Universal Robots PolyScope program: reciprocal_p3_3.urp

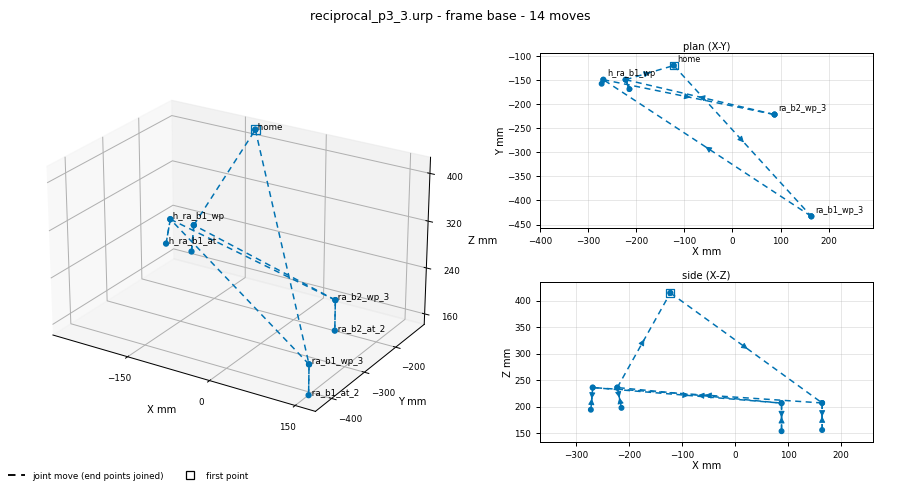
[picture p0: tool path of reciprocal_p3_3.urp in frame base, 14 of 14 moves have a stored position in this frame; points joined in program order, loops and branches not executed]
Program reciprocal_p3_3 (installation=default_1 directory=/programs/../media/urmountpoint_GSJLiG/ITER createdIn=5.3.1.64192 lastSavedIn=5.3.1.64192 robotSerialNumber=20195300365)
Calibrated DH parameters: a=[-0.000093, -0.190649, -0.212673, 0.000091, -0.000205, 0]; d=[0.151591, 44.061648, -42.488068, -1.442789, 0.085322, 0.091911]; alpha=[1.570082, -0.003447, 0.007513, 1.572293, -1.571904, 0]; deltaTheta=[0, -0.672656, 0.728185, -0.055522, 0.000005, 0]
Robot Program (runOnlyOnce=false)
  URCap Gripper Activate (Robotiq_Grippers, Robotiq Inc.) dataModel(ResetAndActivateKey=false)
  URCap Gripper (Robotiq_Grippers, Robotiq Inc.) dataModel(position=50.0, force=100.0, speed=100.0, positionInDouble=50.0, forceInDouble=100.0, speedInDouble=100.0, slaveIds=[9], blocking=true)
  MoveJ speed 60 deg/s, acceleration 80 deg/s^2 (useActiveTCP=true) feature=Base
    Waypoint home: TCP in base x=-122.15 y=-119.32 z=414.454 mm, rx=2.2563 ry=2.1459 rz=-0.0481 rad; joints [-85.681, -56.776, -79.802, -131.025, 89.944, -262.833] deg
  Folder Roof_A
    MoveJ speed 60 deg/s, acceleration 80 deg/s^2 (useActiveTCP=true) feature=Base
      Waypoint ra_b1_wp_3: TCP in base x=164.04 y=-432.993 z=207.005 mm, rx=2.2314 ry=2.1509 rz=0.0059 rad; joints [-53.036, -127.512, -66.191, -73.855, 90.777, -230.696] deg
      Waypoint ra_b1_at_2: TCP in base x=164.049 y=-432.987 z=156.003 mm, rx=2.2314 ry=2.151 rz=0.0059 rad; joints [-53.052, -131.715, -73.279, -62.563, 90.747, -230.647] deg
      URCap Gripper (Robotiq_Grippers, Robotiq Inc.) dataModel(position=100.0, force=100.0, speed=100.0, positionInDouble=100.0, forceInDouble=100.0, speedInDouble=100.0, slaveIds=[9], blocking=true)
      Waypoint ra_b1_wp_4: TCP in base x=164.04 y=-432.993 z=207.005 mm, rx=2.2314 ry=2.1509 rz=0.0059 rad; joints [-53.036, -127.512, -66.191, -73.855, 90.777, -230.696] deg
      Waypoint h_ra_b1_wp: TCP in base x=-268.55 y=-148.787 z=236.04 mm, rx=2.7608 ry=-0.1306 rz=0.0749 rad; joints [-131.096, -88.368, -118.927, -47.1, 105.838, -213.026] deg
      Waypoint h_ra_b1_at: TCP in base x=-272.048 y=-157.193 z=194.251 mm, rx=2.7928 ry=-0.086 rz=0.1068 rad; joints [-130.55, -96.287, -122.586, -37.872, 105.802, -214.66] deg
      URCap Gripper (Robotiq_Grippers, Robotiq Inc.) dataModel(position=50.0, force=100.0, speed=100.0, positionInDouble=50.0, forceInDouble=100.0, speedInDouble=100.0, slaveIds=[9], blocking=true)
      Waypoint h_ra_b1_wp: TCP in base x=-268.55 y=-148.787 z=236.04 mm, rx=2.7608 ry=-0.1306 rz=0.0749 rad; joints [-131.096, -88.368, -118.927, -47.1, 105.838, -213.026] deg
    MoveJ speed 60 deg/s, acceleration 80 deg/s^2 (useActiveTCP=true) feature=Base
      Waypoint ra_b2_wp_3: TCP in base x=87.515 y=-221.249 z=206.702 mm, rx=2.1687 ry=2.2623 rz=-0.0123 rad; joints [-35.23, -70.004, -133.115, -66.455, 89.869, -217.229] deg
      Waypoint ra_b2_at_2: TCP in base x=87.508 y=-221.258 z=153.772 mm, rx=2.1686 ry=2.2623 rz=-0.0124 rad; joints [-35.265, -80.236, -143.583, -45.752, 89.755, -217.149] deg
      URCap Gripper (Robotiq_Grippers, Robotiq Inc.) dataModel(position=100.0, force=100.0, speed=100.0, positionInDouble=100.0, forceInDouble=100.0, speedInDouble=100.0, slaveIds=[9], blocking=true)
      Waypoint ra_b2_wp_4: TCP in base x=87.515 y=-221.249 z=206.702 mm, rx=2.1687 ry=2.2623 rz=-0.0123 rad; joints [-35.23, -70.004, -133.115, -66.455, 89.869, -217.229] deg
      Waypoint h_ra_b2_wp: TCP in base x=-222.173 y=-148.778 z=236.048 mm, rx=2.7617 ry=-0.0717 rz=0.0011 rad; joints [-121.367, -76.176, -130.557, -44.074, 100.878, -206.047] deg
      Waypoint h_ra_b2_at: TCP in base x=-214.314 y=-168.312 z=197.793 mm, rx=2.8721 ry=-0.0559 rz=-0.0607 rad; joints [-115.061, -82.329, -135.249, -37.27, 94.17, -201.737] deg
      URCap Gripper (Robotiq_Grippers, Robotiq Inc.) dataModel(position=50.0, force=100.0, speed=100.0, positionInDouble=50.0, forceInDouble=100.0, speedInDouble=100.0, slaveIds=[9], blocking=true)
      Waypoint h_ra_b2_wp: TCP in base x=-222.173 y=-148.778 z=236.048 mm, rx=2.7617 ry=-0.0717 rz=0.0011 rad; joints [-121.367, -76.176, -130.557, -44.074, 100.878, -206.047] deg
  MoveJ speed 60 deg/s, acceleration 80 deg/s^2 (useActiveTCP=true) feature=Base
    Waypoint home: TCP in base x=-122.15 y=-119.32 z=414.454 mm, rx=2.2563 ry=2.1459 rz=-0.0481 rad; joints [-85.681, -56.776, -79.802, -131.025, 89.944, -262.833] deg
